// TIA Portal V20 export
DATA_BLOCK "SP507"   // DB339
// stored: MemoryReserve 100
   VAR
      "UNWINDER EPCC01 INTERLOCK" : Bool := FALSE;
      "UNWINDER EPCC02 INTERLOCK" : Bool := FALSE;
      "UNWINDER EPCC03 INTERLOCK" : Bool := FALSE;
      "UNWINDER EPCC04 INTERLOCK" : Bool := FALSE;
   END_VAR
BEGIN
END_DATA_BLOCK
